// 取得檔案的參數
TYPE SQL_DxfFileStruct :
STRUCT
	file_Size	: DINT;
	file_data	: ARRAY [0..1048575] OF BYTE;
END_STRUCT
END_TYPE

(* stored: Version 1.1.0.1, ProductVersion 3.1.4026.13
   DUT SQL_DxfFileStruct: Id {dae7dd87-aa1f-4bb8-8b91-f3664882f869} *)
